FUNCTION F_PosnInitial : LREAL
VAR_INPUT
	VeloInit 	: LREAL;
	VeloFinal	: LREAL;
	Accel		: LREAL;
	PosnFinal	: LREAL;
END_VAR
VAR
END_VAR

IF ((2*Accel) + PosnFinal) <> 0 THEN
	F_PosnInitial := ((EXPT(VeloFinal,2) - EXPT(VeloInit,2)) / (2*Accel)) + PosnFinal;
END_IF

END_FUNCTION

(* stored: Version 1.1.0.1
   POU F_PosnInitial: Id {9ecfa6d5-666b-0882-25a3-fae5e0115b35}, SpecialFunc None *)
